PROGRAM PRG_MasterControl
VAR
	eMachineModePrev 	: E_MachineMode := E_MachineMode.STOPPED;
	bModeChanged	 	: BOOL := FALSE;
	bResetStateMachine	: BOOL := FALSE;
	bResetSMDone		: BOOL := FALSE;
	bStoppedResetDone	: BOOL := FALSE;
	
	//Triggers
	rTriggerStopButton	: R_TRIG;
	rTriggerStartButton	: R_TRIG;
	
	//PowerUp Variables
	tonPowerUp				: ton;
	bPowerUpTimerComplete	: BOOL := FALSE;
	bPowerUpDone			: BOOL := FALSE;
	
	//System Initializing Variables
	tonSystemInitialize		: ton;
	rTrigEnterSystemInit 	: R_TRIG;
	bInitResetStarted    	: BOOL := FALSE;
    bInitResetCompleted  	: BOOL := FALSE;
	bSystemInitTimerStart	: BOOL := FALSE;
	bSystemInitReseted		: BOOL := FALSE;

END_VAR

// System Power Up Timer
tonPowerUp( IN 	:= TRUE, 
			PT 	:= T#2S,	
			Q 	=> bPowerUpTimerComplete);

IF bPowerUpTimerComplete AND NOT bPowerUpDone THEN
	GVL_HMI.eMachineMode := E_MachineMode.STOPPED;
	bPowerUpDone := TRUE; // Indicates que the initialization is already happened
END_IF

// Mode Change Monitoring
bModeChanged := (GVL_HMI.eMachineMode <> eMachineModePrev);
eMachineModePrev := GVL_HMI.eMachineMode;

//bResetStateMachine := bModeChanged AND (GVL_HMI.eMachineMode = E_MachineMode.AUTO_CYCLE);

// Buttons Triggers
rTriggerStartButton(CLK := GVL_IO.gDigInputs.bStartButton);
rTriggerStopButton(CLK := GVL_IO.gDigInputs.bStopButton);

//Reset Button Blinking
IF (GVL_HMI.eMachineMode = E_MachineMode.IMEDIATE_FAULT) AND NOT GVL_Safety. bSafetyEnable THEN
	GVL_IO.gDigOutputs.bResetIndicator := GVL_Safety.bResetButtonBlink;
END_IF

// Stop Button monitoring
IF rTriggerStopButton.Q AND NOT (GVL_HMI.eMachineMode = E_MachineMode.SYSTEM_INITIALIZING) THEN
	GVL_HMI.eMachineMode := E_MachineMode.STOPPED;
END_IF

//Safety Enable Monitoring
IF NOT GVL_Safety.bSafetyEnable THEN
	GVL_HMI.eMachineMode := E_MachineMode.IMEDIATE_FAULT;
END_IF

//Reset the Reset flags every time gets out of auto cycle
IF NOT (GVL_HMI.eMachineMode = E_MachineMode.AUTO_CYCLE) THEN
	bResetSMDone := FALSE;
	bResetStateMachine := TRUE;
END_IF

//Resets PRG_SystemIniti *********************************************************************************************
//rTrigEnterSystemInit(CLK := NOT (GVL_HMI.eMachineMode = E_MachineMode.SYSTEM_INITIALIZING));

IF (GVL_HMI.eMachineMode <> E_MachineMode.SYSTEM_INITIALIZING) AND NOT bSystemInitReseted THEN
	bSystemInitReseted := PRG_SystemInit.Reset();
	IF bSystemInitReseted THEN
		bSystemInitTimerStart := FALSE; //Reset timer every time is not in System Initializing
	END_IF
END_IF
//**********************************************************************************************************************
//Reset the Stopped state flags every time gets out of Stopped State
IF NOT (GVL_HMI.eMachineMode = E_MachineMode.STOPPED) THEN
	bStoppedResetDone := PRG_StoppedState.Reset();
END_IF

// Main Master controll logic
CASE GVL_HMI.eMachineMode OF

    E_MachineMode.AUTO_CYCLE: 	// Entry from Stopped state
		IF bResetStateMachine THEN
			bResetSMDone := PRG_StateMachine.Reset(); //Resets the state machine everytime entry this case
		END_IF; 
		
		IF bResetSMDone THEN
			bResetStateMachine := FALSE;
    		PRG_StateMachine(); // calls the state machine
		END_IF

    E_MachineMode.MANUAL:		// Entry from HMI Selection
        PRG_ManualControl(); 

    E_MachineMode.CALIBRATION:	// Entry from HMI Selection
        PRG_Calibration();

        IF PRG_Calibration.bCalibrationFinished THEN
            GVL_HMI.eMachineMode := E_MachineMode.STOPPED;
			PRG_Calibration.Reset(); //TODO
        END_IF

    E_MachineMode.IMEDIATE_FAULT: //Entry from Safety Monitoring
        //PRG_SafetyHandle();

        IF GVL_Safety.bSafetyEnable THEN
            GVL_HMI.eMachineMode := E_MachineMode.SYSTEM_INITIALIZING;
        END_IF

    E_MachineMode.STOPPED:		// Entry from Stop Button or Imediate Fault
        IF bStoppedResetDone THEN
			PRG_StoppedState();
		END_IF
		
        IF rTriggerStartButton.Q AND GVL_Safety.bSafetyEnable AND PRG_StoppedState.bStopAllMotorsDone THEN //only change the state if all motors were stopped
			bStoppedResetDone := FALSE;
            GVL_HMI.eMachineMode := E_MachineMode.SYSTEM_INITIALIZING;
        END_IF
	
	E_MachineMode.SYSTEM_INITIALIZING: // Entry when the machine is first power up to do the homing of the motors
	
       	tonSystemInitialize(IN := bSystemInitTimerStart, PT := T#2S);
		
		bSystemInitReseted := FALSE;
		bSystemInitTimerStart := TRUE;
		
		IF GVL_Safety.bSafetyEnable AND tonSystemInitialize.Q THEN
			PRG_SystemInit(); // Run init procedure
		END_IF
		// Transition to SYSTEM_READY when initialization completes
		IF PRG_SystemInit.bDone AND tonSystemInitialize.Q THEN
			GVL_HMI.eMachineMode := E_MachineMode.SYSTEM_READY;
		END_IF
		
	E_MachineMode.SYSTEM_READY:	// Entry when the start button was pressed on Stop State.
	
		PRG_SystemReady();
		
		IF rTriggerStartButton.Q AND GVL_Safety.bSafetyEnable THEN
			IF NOT GVL_HMI.bIncoherenceDetected THEN
				GVL_HMI.eMachineMode := E_MachineMode.AUTO_CYCLE;
				GVL_HMI.bIncoherenceAlert := FALSE;
			ELSE
				GVL_HMI.bIncoherenceAlert := TRUE;
			END_IF
        END_IF
		
END_CASE

END_PROGRAM

(* stored: Version 1.1.0.1, ProductVersion 3.1.4024.15
   POU PRG_MasterControl: Id {a4cbd161-85e0-4c8d-ae27-b2066d5dd82b}, SpecialFunc None *)
